// TIA Portal V15.1 export
// export: Created 2024-06-21T08:40:51.9562326Z, ExportSetting WithDefaults, DisplayName Totally Integrated Automation Portal, DisplayVersion V15.1 Update 5, DisplayName TIA Portal Openness, DisplayVersion V15.1 Update 5, DisplayName SINAMICS Startdrive Advanced, DisplayVersion V15.1, DisplayName G130, G150, S120, S150, SINAMICS MV, S210, DisplayVersion V15.1, DisplayName G110M, G120, G120C, G120D, G120P, DisplayVersion V15.1, DisplayName STEP 7 Professional, DisplayVersion V15.1 Update 5, DisplayName STEP 7 Safety, DisplayVersion V15.1, DisplayName WinCC Professional, DisplayVersion V15.1 Update 5, DisplayName SIMATIC Visualization Architect, DisplayVersion V15.1
FUNCTION "F209210ZS01Input" : Void   // FC7010, F_FBD
TITLE = Safety Inputs ZMProc / Safety Inputs 209210ZS01
{ S7_Optimized_Access := 'TRUE' }
VERSION : 0.1
// stored: AutoNumber false, IsIECCheckEnabled false, UDAEnableTagReadback false
BEGIN

REGION Network 1: **** 1 - Inputs **** 209210AS10 Reset command Input
   // Reset command Input
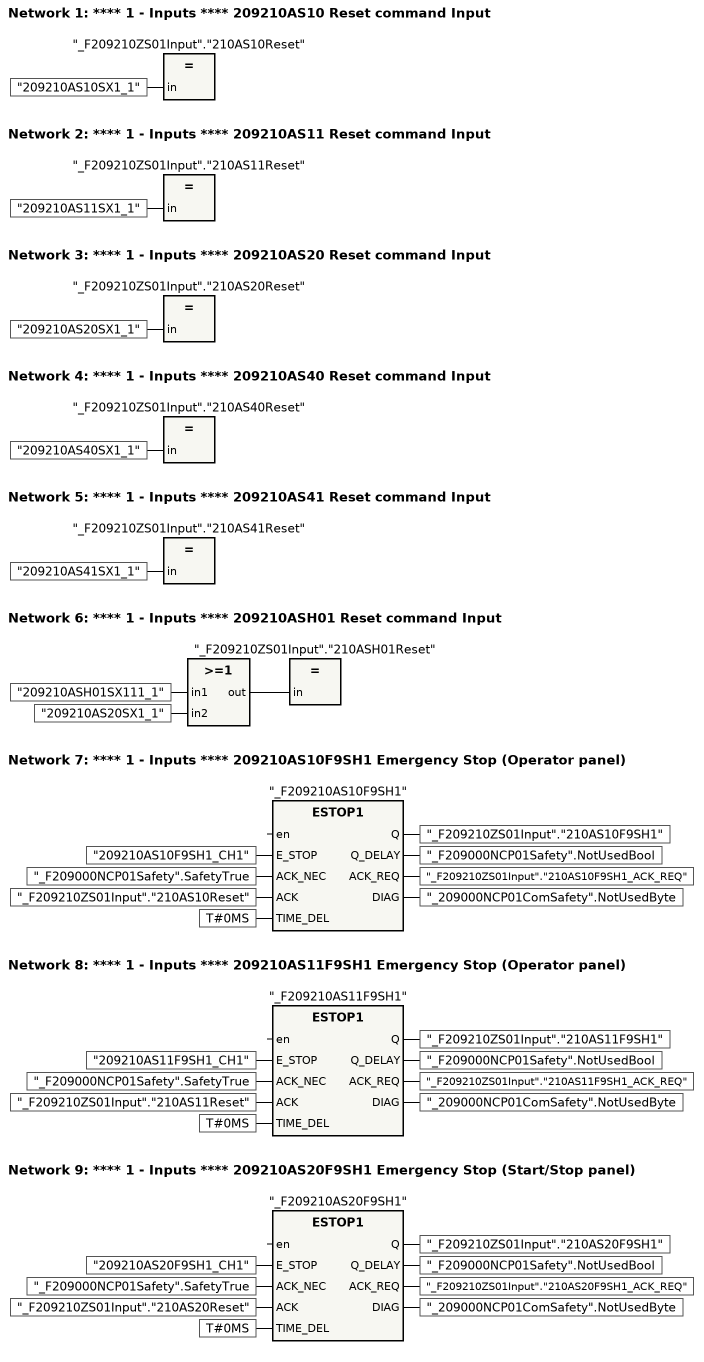
   "_F209210ZS01Input"."210AS10Reset" := "209210AS10SX1_1";
END_REGION

REGION Network 2: **** 1 - Inputs **** 209210AS11 Reset command Input
   // Reset command Input
   "_F209210ZS01Input"."210AS11Reset" := "209210AS11SX1_1";
END_REGION

REGION Network 3: **** 1 - Inputs **** 209210AS20 Reset command Input
   // Reset command Input
   "_F209210ZS01Input"."210AS20Reset" := "209210AS20SX1_1";
END_REGION

REGION Network 4: **** 1 - Inputs **** 209210AS40 Reset command Input
   // Reset command Input
   "_F209210ZS01Input"."210AS40Reset" := "209210AS40SX1_1";
END_REGION

REGION Network 5: **** 1 - Inputs **** 209210AS41 Reset command Input
   // Reset command Input
   "_F209210ZS01Input"."210AS41Reset" := "209210AS41SX1_1";
END_REGION

REGION Network 6: **** 1 - Inputs **** 209210ASH01 Reset command Input
   // Reset command Input
   "_F209210ZS01Input"."210ASH01Reset" := "209210ASH01SX111_1" OR "209210AS20SX1_1";
END_REGION

REGION Network 7: **** 1 - Inputs **** 209210AS10F9SH1 Emergency Stop (Operator panel)
   // Emergency Stop
   "_F209210AS10F9SH1"(E_STOP := "209210AS10F9SH1_CH1",   // ESTOP1
                       ACK_NEC := "_F209000NCP01Safety".SafetyTrue,
                       ACK := "_F209210ZS01Input"."210AS10Reset",
                       TIME_DEL := T#0MS,
                       Q => "_F209210ZS01Input"."210AS10F9SH1",
                       Q_DELAY => "_F209000NCP01Safety".NotUsedBool,
                       ACK_REQ => "_F209210ZS01Input"."210AS10F9SH1_ACK_REQ",
                       DIAG => "_209000NCP01ComSafety".NotUsedByte);
END_REGION

REGION Network 8: **** 1 - Inputs **** 209210AS11F9SH1 Emergency Stop (Operator panel)
   // Emergency Stop
   "_F209210AS11F9SH1"(E_STOP := "209210AS11F9SH1_CH1",   // ESTOP1
                       ACK_NEC := "_F209000NCP01Safety".SafetyTrue,
                       ACK := "_F209210ZS01Input"."210AS11Reset",
                       TIME_DEL := T#0MS,
                       Q => "_F209210ZS01Input"."210AS11F9SH1",
                       Q_DELAY => "_F209000NCP01Safety".NotUsedBool,
                       ACK_REQ => "_F209210ZS01Input"."210AS11F9SH1_ACK_REQ",
                       DIAG => "_209000NCP01ComSafety".NotUsedByte);
END_REGION

REGION Network 9: **** 1 - Inputs **** 209210AS20F9SH1 Emergency Stop (Start/Stop panel)
   // Emergency Stop
   "_F209210AS20F9SH1"(E_STOP := "209210AS20F9SH1_CH1",   // ESTOP1
                       ACK_NEC := "_F209000NCP01Safety".SafetyTrue,
                       ACK := "_F209210ZS01Input"."210AS20Reset",
                       TIME_DEL := T#0MS,
                       Q => "_F209210ZS01Input"."210AS20F9SH1",
                       Q_DELAY => "_F209000NCP01Safety".NotUsedBool,
                       ACK_REQ => "_F209210ZS01Input"."210AS20F9SH1_ACK_REQ",
                       DIAG => "_209000NCP01ComSafety".NotUsedByte);
END_REGION

REGION Network 10: **** 1 - Inputs **** 209210AS40F9SH1 Emergency Stop (External panel)
   // Emergency Stop
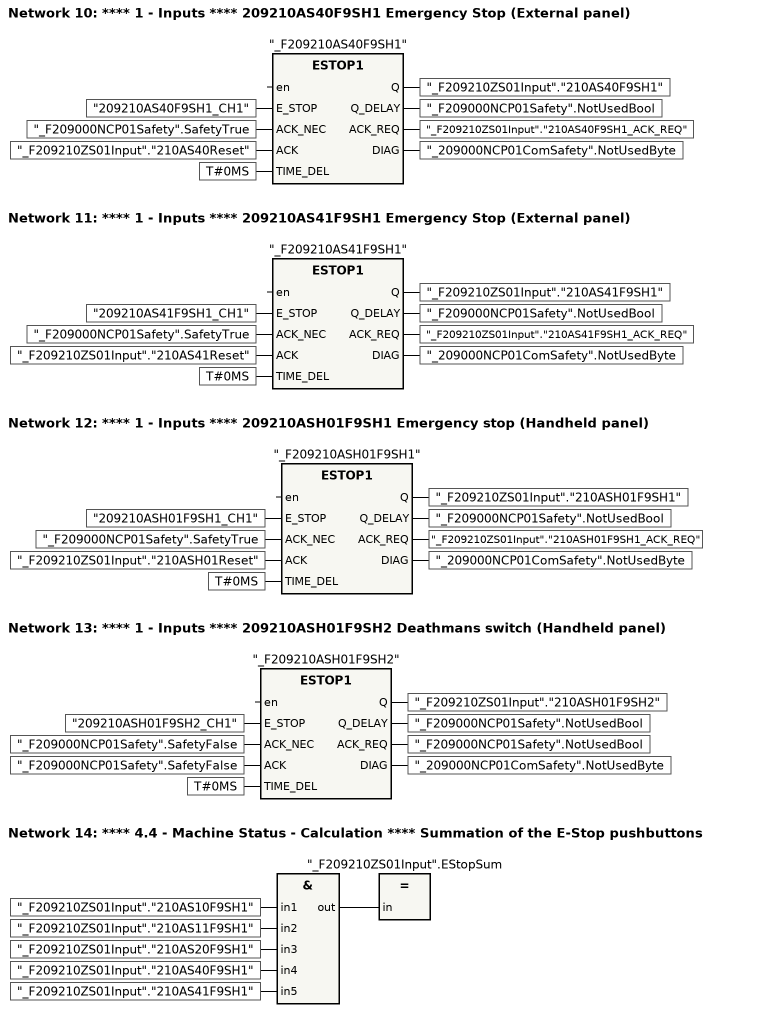
   "_F209210AS40F9SH1"(E_STOP := "209210AS40F9SH1_CH1",   // ESTOP1
                       ACK_NEC := "_F209000NCP01Safety".SafetyTrue,
                       ACK := "_F209210ZS01Input"."210AS40Reset",
                       TIME_DEL := T#0MS,
                       Q => "_F209210ZS01Input"."210AS40F9SH1",
                       Q_DELAY => "_F209000NCP01Safety".NotUsedBool,
                       ACK_REQ => "_F209210ZS01Input"."210AS40F9SH1_ACK_REQ",
                       DIAG => "_209000NCP01ComSafety".NotUsedByte);
END_REGION

REGION Network 11: **** 1 - Inputs **** 209210AS41F9SH1 Emergency Stop (External panel)
   // Emergency Stop
   "_F209210AS41F9SH1"(E_STOP := "209210AS41F9SH1_CH1",   // ESTOP1
                       ACK_NEC := "_F209000NCP01Safety".SafetyTrue,
                       ACK := "_F209210ZS01Input"."210AS41Reset",
                       TIME_DEL := T#0MS,
                       Q => "_F209210ZS01Input"."210AS41F9SH1",
                       Q_DELAY => "_F209000NCP01Safety".NotUsedBool,
                       ACK_REQ => "_F209210ZS01Input"."210AS41F9SH1_ACK_REQ",
                       DIAG => "_209000NCP01ComSafety".NotUsedByte);
END_REGION

REGION Network 12: **** 1 - Inputs **** 209210ASH01F9SH1 Emergency stop (Handheld panel)
   // Emergency Stop
   "_F209210ASH01F9SH1"(E_STOP := "209210ASH01F9SH1_CH1",   // ESTOP1
                        ACK_NEC := "_F209000NCP01Safety".SafetyTrue,
                        ACK := "_F209210ZS01Input"."210ASH01Reset",
                        TIME_DEL := T#0MS,
                        Q => "_F209210ZS01Input"."210ASH01F9SH1",
                        Q_DELAY => "_F209000NCP01Safety".NotUsedBool,
                        ACK_REQ => "_F209210ZS01Input"."210ASH01F9SH1_ACK_REQ",
                        DIAG => "_209000NCP01ComSafety".NotUsedByte);
END_REGION

REGION Network 13: **** 1 - Inputs **** 209210ASH01F9SH2 Deathmans switch (Handheld panel)
   // Emergency Stop
   "_F209210ASH01F9SH2"(E_STOP := "209210ASH01F9SH2_CH1",   // ESTOP1
                        ACK_NEC := "_F209000NCP01Safety".SafetyFalse,
                        ACK := "_F209000NCP01Safety".SafetyFalse,
                        TIME_DEL := T#0MS,
                        Q => "_F209210ZS01Input"."210ASH01F9SH2",
                        Q_DELAY => "_F209000NCP01Safety".NotUsedBool,
                        ACK_REQ => "_F209000NCP01Safety".NotUsedBool,
                        DIAG => "_209000NCP01ComSafety".NotUsedByte);
END_REGION

REGION Network 14: **** 4.4 - Machine Status - Calculation **** Summation of the E-Stop pushbuttons
   // Summation of the E-Stop pushbuttons
   "_F209210ZS01Input".EStopSum := "_F209210ZS01Input"."210AS10F9SH1" AND "_F209210ZS01Input"."210AS11F9SH1" AND "_F209210ZS01Input"."210AS20F9SH1" AND "_F209210ZS01Input"."210AS40F9SH1" AND "_F209210ZS01Input"."210AS41F9SH1";
END_REGION
END_FUNCTION
